(* IEC 61131-3 sources: AXOpen/src/core/ctrl/src/IxUtilities, 5 files *)

(* ---- IxCRC_16.st ---- *)
USING System.Strings;
USING System.SerDe;

NAMESPACE ix.framework.core
    FUNCTION PUBLIC IxCRC_16 : WORD
		VAR_INPUT
			In : STRING[254];
		END_VAR
		VAR
			crc : WORD := WORD#16#FFFF;
			i : UINT;
			maxIndex : UINT;
			serialized : ARRAY[0..255] OF BYTE;
		END_VAR
		VAR
			//Precalculated values for polynomial generator of value 0x1021
			CRC_TABLE : ARRAY[0..255] OF WORD := [
				WORD#16#0000, WORD#16#1021, WORD#16#2042, WORD#16#3063, WORD#16#4084, WORD#16#50A5, WORD#16#60C6, WORD#16#70E7, WORD#16#8108, WORD#16#9129, WORD#16#A14A, WORD#16#B16B, WORD#16#C18C, WORD#16#D1AD, WORD#16#E1CE, WORD#16#F1EF,
				WORD#16#1231, WORD#16#0210, WORD#16#3273, WORD#16#2252, WORD#16#52B5, WORD#16#4294, WORD#16#72F7, WORD#16#62D6, WORD#16#9339, WORD#16#8318, WORD#16#B37B, WORD#16#A35A, WORD#16#D3BD, WORD#16#C39C, WORD#16#F3FF, WORD#16#E3DE,
				WORD#16#2462, WORD#16#3443, WORD#16#0420, WORD#16#1401, WORD#16#64E6, WORD#16#74C7, WORD#16#44A4, WORD#16#5485, WORD#16#A56A, WORD#16#B54B, WORD#16#8528, WORD#16#9509, WORD#16#E5EE, WORD#16#F5CF, WORD#16#C5AC, WORD#16#D58D,
				WORD#16#3653, WORD#16#2672, WORD#16#1611, WORD#16#0630, WORD#16#76D7, WORD#16#66F6, WORD#16#5695, WORD#16#46B4, WORD#16#B75B, WORD#16#A77A, WORD#16#9719, WORD#16#8738, WORD#16#F7DF, WORD#16#E7FE, WORD#16#D79D, WORD#16#C7BC,
				WORD#16#48C4, WORD#16#58E5, WORD#16#6886, WORD#16#78A7, WORD#16#0840, WORD#16#1861, WORD#16#2802, WORD#16#3823, WORD#16#C9CC, WORD#16#D9ED, WORD#16#E98E, WORD#16#F9AF, WORD#16#8948, WORD#16#9969, WORD#16#A90A, WORD#16#B92B,
				WORD#16#5AF5, WORD#16#4AD4, WORD#16#7AB7, WORD#16#6A96, WORD#16#1A71, WORD#16#0A50, WORD#16#3A33, WORD#16#2A12, WORD#16#DBFD, WORD#16#CBDC, WORD#16#FBBF, WORD#16#EB9E, WORD#16#9B79, WORD#16#8B58, WORD#16#BB3B, WORD#16#AB1A,
				WORD#16#6CA6, WORD#16#7C87, WORD#16#4CE4, WORD#16#5CC5, WORD#16#2C22, WORD#16#3C03, WORD#16#0C60, WORD#16#1C41, WORD#16#EDAE, WORD#16#FD8F, WORD#16#CDEC, WORD#16#DDCD, WORD#16#AD2A, WORD#16#BD0B, WORD#16#8D68, WORD#16#9D49,
				WORD#16#7E97, WORD#16#6EB6, WORD#16#5ED5, WORD#16#4EF4, WORD#16#3E13, WORD#16#2E32, WORD#16#1E51, WORD#16#0E70, WORD#16#FF9F, WORD#16#EFBE, WORD#16#DFDD, WORD#16#CFFC, WORD#16#BF1B, WORD#16#AF3A, WORD#16#9F59, WORD#16#8F78,
				WORD#16#9188, WORD#16#81A9, WORD#16#B1CA, WORD#16#A1EB, WORD#16#D10C, WORD#16#C12D, WORD#16#F14E, WORD#16#E16F, WORD#16#1080, WORD#16#00A1, WORD#16#30C2, WORD#16#20E3, WORD#16#5004, WORD#16#4025, WORD#16#7046, WORD#16#6067,
				WORD#16#83B9, WORD#16#9398, WORD#16#A3FB, WORD#16#B3DA, WORD#16#C33D, WORD#16#D31C, WORD#16#E37F, WORD#16#F35E, WORD#16#02B1, WORD#16#1290, WORD#16#22F3, WORD#16#32D2, WORD#16#4235, WORD#16#5214, WORD#16#6277, WORD#16#7256,
				WORD#16#B5EA, WORD#16#A5CB, WORD#16#95A8, WORD#16#8589, WORD#16#F56E, WORD#16#E54F, WORD#16#D52C, WORD#16#C50D, WORD#16#34E2, WORD#16#24C3, WORD#16#14A0, WORD#16#0481, WORD#16#7466, WORD#16#6447, WORD#16#5424, WORD#16#4405,
				WORD#16#A7DB, WORD#16#B7FA, WORD#16#8799, WORD#16#97B8, WORD#16#E75F, WORD#16#F77E, WORD#16#C71D, WORD#16#D73C, WORD#16#26D3, WORD#16#36F2, WORD#16#0691, WORD#16#16B0, WORD#16#6657, WORD#16#7676, WORD#16#4615, WORD#16#5634,
				WORD#16#D94C, WORD#16#C96D, WORD#16#F90E, WORD#16#E92F, WORD#16#99C8, WORD#16#89E9, WORD#16#B98A, WORD#16#A9AB, WORD#16#5844, WORD#16#4865, WORD#16#7806, WORD#16#6827, WORD#16#18C0, WORD#16#08E1, WORD#16#3882, WORD#16#28A3,
				WORD#16#CB7D, WORD#16#DB5C, WORD#16#EB3F, WORD#16#FB1E, WORD#16#8BF9, WORD#16#9BD8, WORD#16#ABBB, WORD#16#BB9A, WORD#16#4A75, WORD#16#5A54, WORD#16#6A37, WORD#16#7A16, WORD#16#0AF1, WORD#16#1AD0, WORD#16#2AB3, WORD#16#3A92,
				WORD#16#FD2E, WORD#16#ED0F, WORD#16#DD6C, WORD#16#CD4D, WORD#16#BDAA, WORD#16#AD8B, WORD#16#9DE8, WORD#16#8DC9, WORD#16#7C26, WORD#16#6C07, WORD#16#5C64, WORD#16#4C45, WORD#16#3CA2, WORD#16#2C83, WORD#16#1CE0, WORD#16#0CC1,
				WORD#16#EF1F, WORD#16#FF3E, WORD#16#CF5D, WORD#16#DF7C, WORD#16#AF9B, WORD#16#BFBA, WORD#16#8FD9, WORD#16#9FF8, WORD#16#6E17, WORD#16#7E36, WORD#16#4E55, WORD#16#5E74, WORD#16#2E93, WORD#16#3EB2, WORD#16#0ED1, WORD#16#1EF0];
		END_VAR
		IxCRC_16 := crc;

		maxIndex := UINT#0;

		maxIndex := Serialize(UINT#0, In, serialized,System.SerDe.Endianness#Little) - UINT#1;

		IF maxIndex < UINT#1 THEN
			RETURN;
		END_IF;

		FOR i := UINT#1 TO maxIndex BY UINT#1 DO
			// crc := SHL(crc, 8) XOR CRC_TABLE[SHR(crc, 8) XOR bByte];
			crc := ixXor(SHL(crc, UINT#8),CRC_TABLE[TO_INT(ixXor(SHR(crc, UINT#8) , serialized[i]))]);
		END_FOR;

		IxCRC_16 := crc;
    END_FUNCTION
END_NAMESPACE

(* ---- IxCRC_32.st ---- *)
USING System.Strings;
USING System.SerDe;

NAMESPACE ix.framework.core
    FUNCTION PUBLIC IxCRC_32 : DWORD
		VAR_INPUT
			In : STRING[254];
		END_VAR
		VAR
			crc : DWORD := DWORD#16#FFFFFFFF;
			i : UINT;
			maxIndex : UINT;
			serialized : ARRAY[0..255] OF BYTE;
		END_VAR
		VAR
			//Precalculated values for polynomial generator of value 0x04C11DB7
			CRC_TABLE : ARRAY[0..255] OF DWORD := [
				DWORD#16#00000000, DWORD#16#04C11DB7, DWORD#16#09823B6E, DWORD#16#0D4326D9, DWORD#16#130476DC, DWORD#16#17C56B6B, DWORD#16#1A864DB2, DWORD#16#1E475005, DWORD#16#2608EDB8, DWORD#16#22C9F00F, DWORD#16#2F8AD6D6, DWORD#16#2B4BCB61, DWORD#16#350C9B64, DWORD#16#31CD86D3, DWORD#16#3C8EA00A, DWORD#16#384FBDBD,
				DWORD#16#4C11DB70, DWORD#16#48D0C6C7, DWORD#16#4593E01E, DWORD#16#4152FDA9, DWORD#16#5F15ADAC, DWORD#16#5BD4B01B, DWORD#16#569796C2, DWORD#16#52568B75, DWORD#16#6A1936C8, DWORD#16#6ED82B7F, DWORD#16#639B0DA6, DWORD#16#675A1011, DWORD#16#791D4014, DWORD#16#7DDC5DA3, DWORD#16#709F7B7A, DWORD#16#745E66CD,
				DWORD#16#9823B6E0, DWORD#16#9CE2AB57, DWORD#16#91A18D8E, DWORD#16#95609039, DWORD#16#8B27C03C, DWORD#16#8FE6DD8B, DWORD#16#82A5FB52, DWORD#16#8664E6E5, DWORD#16#BE2B5B58, DWORD#16#BAEA46EF, DWORD#16#B7A96036, DWORD#16#B3687D81, DWORD#16#AD2F2D84, DWORD#16#A9EE3033, DWORD#16#A4AD16EA, DWORD#16#A06C0B5D,
				DWORD#16#D4326D90, DWORD#16#D0F37027, DWORD#16#DDB056FE, DWORD#16#D9714B49, DWORD#16#C7361B4C, DWORD#16#C3F706FB, DWORD#16#CEB42022, DWORD#16#CA753D95, DWORD#16#F23A8028, DWORD#16#F6FB9D9F, DWORD#16#FBB8BB46, DWORD#16#FF79A6F1, DWORD#16#E13EF6F4, DWORD#16#E5FFEB43, DWORD#16#E8BCCD9A, DWORD#16#EC7DD02D,
				DWORD#16#34867077, DWORD#16#30476DC0, DWORD#16#3D044B19, DWORD#16#39C556AE, DWORD#16#278206AB, DWORD#16#23431B1C, DWORD#16#2E003DC5, DWORD#16#2AC12072, DWORD#16#128E9DCF, DWORD#16#164F8078, DWORD#16#1B0CA6A1, DWORD#16#1FCDBB16, DWORD#16#018AEB13, DWORD#16#054BF6A4, DWORD#16#0808D07D, DWORD#16#0CC9CDCA,
				DWORD#16#7897AB07, DWORD#16#7C56B6B0, DWORD#16#71159069, DWORD#16#75D48DDE, DWORD#16#6B93DDDB, DWORD#16#6F52C06C, DWORD#16#6211E6B5, DWORD#16#66D0FB02, DWORD#16#5E9F46BF, DWORD#16#5A5E5B08, DWORD#16#571D7DD1, DWORD#16#53DC6066, DWORD#16#4D9B3063, DWORD#16#495A2DD4, DWORD#16#44190B0D, DWORD#16#40D816BA,
				DWORD#16#ACA5C697, DWORD#16#A864DB20, DWORD#16#A527FDF9, DWORD#16#A1E6E04E, DWORD#16#BFA1B04B, DWORD#16#BB60ADFC, DWORD#16#B6238B25, DWORD#16#B2E29692, DWORD#16#8AAD2B2F, DWORD#16#8E6C3698, DWORD#16#832F1041, DWORD#16#87EE0DF6, DWORD#16#99A95DF3, DWORD#16#9D684044, DWORD#16#902B669D, DWORD#16#94EA7B2A,
				DWORD#16#E0B41DE7, DWORD#16#E4750050, DWORD#16#E9362689, DWORD#16#EDF73B3E, DWORD#16#F3B06B3B, DWORD#16#F771768C, DWORD#16#FA325055, DWORD#16#FEF34DE2, DWORD#16#C6BCF05F, DWORD#16#C27DEDE8, DWORD#16#CF3ECB31, DWORD#16#CBFFD686, DWORD#16#D5B88683, DWORD#16#D1799B34, DWORD#16#DC3ABDED, DWORD#16#D8FBA05A,
				DWORD#16#690CE0EE, DWORD#16#6DCDFD59, DWORD#16#608EDB80, DWORD#16#644FC637, DWORD#16#7A089632, DWORD#16#7EC98B85, DWORD#16#738AAD5C, DWORD#16#774BB0EB, DWORD#16#4F040D56, DWORD#16#4BC510E1, DWORD#16#46863638, DWORD#16#42472B8F, DWORD#16#5C007B8A, DWORD#16#58C1663D, DWORD#16#558240E4, DWORD#16#51435D53,
				DWORD#16#251D3B9E, DWORD#16#21DC2629, DWORD#16#2C9F00F0, DWORD#16#285E1D47, DWORD#16#36194D42, DWORD#16#32D850F5, DWORD#16#3F9B762C, DWORD#16#3B5A6B9B, DWORD#16#0315D626, DWORD#16#07D4CB91, DWORD#16#0A97ED48, DWORD#16#0E56F0FF, DWORD#16#1011A0FA, DWORD#16#14D0BD4D, DWORD#16#19939B94, DWORD#16#1D528623,
				DWORD#16#F12F560E, DWORD#16#F5EE4BB9, DWORD#16#F8AD6D60, DWORD#16#FC6C70D7, DWORD#16#E22B20D2, DWORD#16#E6EA3D65, DWORD#16#EBA91BBC, DWORD#16#EF68060B, DWORD#16#D727BBB6, DWORD#16#D3E6A601, DWORD#16#DEA580D8, DWORD#16#DA649D6F, DWORD#16#C423CD6A, DWORD#16#C0E2D0DD, DWORD#16#CDA1F604, DWORD#16#C960EBB3,
				DWORD#16#BD3E8D7E, DWORD#16#B9FF90C9, DWORD#16#B4BCB610, DWORD#16#B07DABA7, DWORD#16#AE3AFBA2, DWORD#16#AAFBE615, DWORD#16#A7B8C0CC, DWORD#16#A379DD7B, DWORD#16#9B3660C6, DWORD#16#9FF77D71, DWORD#16#92B45BA8, DWORD#16#9675461F, DWORD#16#8832161A, DWORD#16#8CF30BAD, DWORD#16#81B02D74, DWORD#16#857130C3,
				DWORD#16#5D8A9099, DWORD#16#594B8D2E, DWORD#16#5408ABF7, DWORD#16#50C9B640, DWORD#16#4E8EE645, DWORD#16#4A4FFBF2, DWORD#16#470CDD2B, DWORD#16#43CDC09C, DWORD#16#7B827D21, DWORD#16#7F436096, DWORD#16#7200464F, DWORD#16#76C15BF8, DWORD#16#68860BFD, DWORD#16#6C47164A, DWORD#16#61043093, DWORD#16#65C52D24,
				DWORD#16#119B4BE9, DWORD#16#155A565E, DWORD#16#18197087, DWORD#16#1CD86D30, DWORD#16#029F3D35, DWORD#16#065E2082, DWORD#16#0B1D065B, DWORD#16#0FDC1BEC, DWORD#16#3793A651, DWORD#16#3352BBE6, DWORD#16#3E119D3F, DWORD#16#3AD08088, DWORD#16#2497D08D, DWORD#16#2056CD3A, DWORD#16#2D15EBE3, DWORD#16#29D4F654,
				DWORD#16#C5A92679, DWORD#16#C1683BCE, DWORD#16#CC2B1D17, DWORD#16#C8EA00A0, DWORD#16#D6AD50A5, DWORD#16#D26C4D12, DWORD#16#DF2F6BCB, DWORD#16#DBEE767C, DWORD#16#E3A1CBC1, DWORD#16#E760D676, DWORD#16#EA23F0AF, DWORD#16#EEE2ED18, DWORD#16#F0A5BD1D, DWORD#16#F464A0AA, DWORD#16#F9278673, DWORD#16#FDE69BC4,
				DWORD#16#89B8FD09, DWORD#16#8D79E0BE, DWORD#16#803AC667, DWORD#16#84FBDBD0, DWORD#16#9ABC8BD5, DWORD#16#9E7D9662, DWORD#16#933EB0BB, DWORD#16#97FFAD0C, DWORD#16#AFB010B1, DWORD#16#AB710D06, DWORD#16#A6322BDF, DWORD#16#A2F33668, DWORD#16#BCB4666D, DWORD#16#B8757BDA, DWORD#16#B5365D03, DWORD#16#B1F740B4];
		END_VAR
		IxCRC_32 := crc;

		maxIndex := UINT#0;

		maxIndex := Serialize(UINT#0, In, serialized,System.SerDe.Endianness#Little) - UINT#1;

		IF maxIndex < UINT#1 THEN
			RETURN;
		END_IF;

		FOR i := UINT#1 TO maxIndex BY UINT#1 DO
			// posD := SHR(crc, 24) XOR bByte;
			// pos := UDINT_TO_BYTE(posD);

			// crc := SHL(crc, 8) XOR CRC_TABLE[pos];

			crc := ixXor(SHL(crc, UINT#8),CRC_TABLE[TO_INT(ixXor(SHR(crc, UINT#24) , serialized[i]))]);
		END_FOR;

		IxCRC_32 := crc;
    END_FUNCTION
END_NAMESPACE

(* ---- IxCRC_8.st ---- *)
USING System.Strings;
USING System.SerDe;

NAMESPACE ix.framework.core
    FUNCTION PUBLIC IxCRC_8 : BYTE
		VAR_INPUT
			In : STRING[254];
		END_VAR
		VAR
			crc : BYTE := BYTE#16#FF;
			i : UINT;
			maxIndex : UINT;
			serialized : ARRAY[0..255] OF BYTE;
		END_VAR
		VAR
			//Precalculated values for polynomial generator of value 0x1D
			CRC_TABLE : ARRAY[0..255] OF BYTE := [
				BYTE#16#00,	BYTE#16#1D,	BYTE#16#3A,	BYTE#16#27,	BYTE#16#74,	BYTE#16#69,	BYTE#16#4E,	BYTE#16#53,	BYTE#16#E8,	BYTE#16#F5,	BYTE#16#D2,	BYTE#16#CF,	BYTE#16#9C,	BYTE#16#81,	BYTE#16#A6,	BYTE#16#BB,
				BYTE#16#CD,	BYTE#16#D0,	BYTE#16#F7,	BYTE#16#EA,	BYTE#16#B9,	BYTE#16#A4,	BYTE#16#83,	BYTE#16#9E,	BYTE#16#25,	BYTE#16#38,	BYTE#16#1F,	BYTE#16#02,	BYTE#16#51,	BYTE#16#4C,	BYTE#16#6B,	BYTE#16#76,
				BYTE#16#87,	BYTE#16#9A,	BYTE#16#BD,	BYTE#16#A0,	BYTE#16#F3,	BYTE#16#EE,	BYTE#16#C9,	BYTE#16#D4,	BYTE#16#6F,	BYTE#16#72,	BYTE#16#55,	BYTE#16#48,	BYTE#16#1B,	BYTE#16#06,	BYTE#16#21,	BYTE#16#3C,
				BYTE#16#4A,	BYTE#16#57,	BYTE#16#70,	BYTE#16#6D,	BYTE#16#3E,	BYTE#16#23,	BYTE#16#04,	BYTE#16#19,	BYTE#16#A2,	BYTE#16#BF,	BYTE#16#98,	BYTE#16#85,	BYTE#16#D6,	BYTE#16#CB,	BYTE#16#EC,	BYTE#16#F1,
				BYTE#16#13,	BYTE#16#0E,	BYTE#16#29,	BYTE#16#34,	BYTE#16#67,	BYTE#16#7A,	BYTE#16#5D,	BYTE#16#40,	BYTE#16#FB,	BYTE#16#E6,	BYTE#16#C1,	BYTE#16#DC,	BYTE#16#8F,	BYTE#16#92,	BYTE#16#B5,	BYTE#16#A8,
				BYTE#16#DE,	BYTE#16#C3,	BYTE#16#E4,	BYTE#16#F9,	BYTE#16#AA,	BYTE#16#B7,	BYTE#16#90,	BYTE#16#8D,	BYTE#16#36,	BYTE#16#2B,	BYTE#16#0C,	BYTE#16#11,	BYTE#16#42,	BYTE#16#5F,	BYTE#16#78,	BYTE#16#65,
				BYTE#16#94,	BYTE#16#89,	BYTE#16#AE,	BYTE#16#B3,	BYTE#16#E0,	BYTE#16#FD,	BYTE#16#DA,	BYTE#16#C7,	BYTE#16#7C,	BYTE#16#61,	BYTE#16#46,	BYTE#16#5B,	BYTE#16#08,	BYTE#16#15,	BYTE#16#32,	BYTE#16#2F,
				BYTE#16#59,	BYTE#16#44,	BYTE#16#63,	BYTE#16#7E,	BYTE#16#2D,	BYTE#16#30,	BYTE#16#17,	BYTE#16#0A,	BYTE#16#B1,	BYTE#16#AC,	BYTE#16#8B,	BYTE#16#96,	BYTE#16#C5,	BYTE#16#D8,	BYTE#16#FF,	BYTE#16#E2,
				BYTE#16#26,	BYTE#16#3B,	BYTE#16#1C,	BYTE#16#01,	BYTE#16#52,	BYTE#16#4F,	BYTE#16#68,	BYTE#16#75,	BYTE#16#CE,	BYTE#16#D3,	BYTE#16#F4,	BYTE#16#E9,	BYTE#16#BA,	BYTE#16#A7,	BYTE#16#80,	BYTE#16#9D,
				BYTE#16#EB,	BYTE#16#F6,	BYTE#16#D1,	BYTE#16#CC,	BYTE#16#9F,	BYTE#16#82,	BYTE#16#A5,	BYTE#16#B8,	BYTE#16#03,	BYTE#16#1E,	BYTE#16#39,	BYTE#16#24,	BYTE#16#77,	BYTE#16#6A,	BYTE#16#4D,	BYTE#16#50,
				BYTE#16#A1,	BYTE#16#BC,	BYTE#16#9B,	BYTE#16#86,	BYTE#16#D5,	BYTE#16#C8,	BYTE#16#EF,	BYTE#16#F2,	BYTE#16#49,	BYTE#16#54,	BYTE#16#73,	BYTE#16#6E,	BYTE#16#3D,	BYTE#16#20,	BYTE#16#07,	BYTE#16#1A,
				BYTE#16#6C,	BYTE#16#71,	BYTE#16#56,	BYTE#16#4B,	BYTE#16#18,	BYTE#16#05,	BYTE#16#22,	BYTE#16#3F,	BYTE#16#84,	BYTE#16#99,	BYTE#16#BE,	BYTE#16#A3,	BYTE#16#F0,	BYTE#16#ED,	BYTE#16#CA,	BYTE#16#D7,
				BYTE#16#35,	BYTE#16#28,	BYTE#16#0F,	BYTE#16#12,	BYTE#16#41,	BYTE#16#5C,	BYTE#16#7B,	BYTE#16#66,	BYTE#16#DD,	BYTE#16#C0,	BYTE#16#E7,	BYTE#16#FA,	BYTE#16#A9,	BYTE#16#B4,	BYTE#16#93,	BYTE#16#8E,
				BYTE#16#F8,	BYTE#16#E5,	BYTE#16#C2,	BYTE#16#DF,	BYTE#16#8C,	BYTE#16#91,	BYTE#16#B6,	BYTE#16#AB,	BYTE#16#10,	BYTE#16#0D,	BYTE#16#2A,	BYTE#16#37,	BYTE#16#64,	BYTE#16#79,	BYTE#16#5E,	BYTE#16#43,
				BYTE#16#B2,	BYTE#16#AF,	BYTE#16#88,	BYTE#16#95,	BYTE#16#C6,	BYTE#16#DB,	BYTE#16#FC,	BYTE#16#E1,	BYTE#16#5A,	BYTE#16#47,	BYTE#16#60,	BYTE#16#7D,	BYTE#16#2E,	BYTE#16#33,	BYTE#16#14,	BYTE#16#09,
				BYTE#16#7F,	BYTE#16#62,	BYTE#16#45,	BYTE#16#58,	BYTE#16#0B,	BYTE#16#16,	BYTE#16#31,	BYTE#16#2C,	BYTE#16#97,	BYTE#16#8A,	BYTE#16#AD,	BYTE#16#B0,	BYTE#16#E3,	BYTE#16#FE,	BYTE#16#D9,	BYTE#16#C4];
		END_VAR
		IxCRC_8 := crc;

		maxIndex := UINT#0;

		maxIndex := Serialize(UINT#0, In, serialized, System.SerDe.Endianness#Little) - UINT#1;

		IF maxIndex < UINT#1 THEN
			RETURN;
		END_IF;

		FOR i := UINT#1 TO maxIndex BY UINT#1 DO
			//crc := CRC_TABLE[bByte XOR crc];
			crc := CRC_TABLE[TO_INT(ixXor(crc , TO_BYTE(TO_CHAR(serialized[i]))))];
		END_FOR;
		IxCRC_8 := crc;
    END_FUNCTION
END_NAMESPACE

(* ---- XORs.st ---- *)
// USING System.BitAccess;

NAMESPACE ix.framework.core
    FUNCTION ixXor : BYTE
        VAR_INPUT
            In1 : BYTE;
            In2 : BYTE;
        END_VAR
        VAR_TEMP
            retval : BYTE;
            i : USINT;
        END_VAR
        retval := BYTE#0;

        // TODO check the performance of both principles
        // FOR i := USINT#0 TO USINT#7 DO
        //     SetBit(retval,i,GetBit(In1,i) XOR GetBit(In2,i));
        // END_FOR;

        retval.%X0 := In1.%X0  XOR In2.%X0 ;
        retval.%X1 := In1.%X1  XOR In2.%X1 ;
        retval.%X2 := In1.%X2  XOR In2.%X2 ;
        retval.%X3 := In1.%X3  XOR In2.%X3 ;
        retval.%X4 := In1.%X4  XOR In2.%X4 ;
        retval.%X5 := In1.%X5  XOR In2.%X5 ;
        retval.%X6 := In1.%X6  XOR In2.%X6 ;
        retval.%X7 := In1.%X7  XOR In2.%X7 ;

        ixXor := retval;
    END_FUNCTION

    FUNCTION ixXor : WORD
        VAR_INPUT
            In1 : WORD;
            In2 : WORD;
        END_VAR
        VAR_TEMP
            retval : WORD;
            i : USINT;
        END_VAR
        retval := WORD#0;

        // TODO check the performance of both principles
        // FOR i := USINT#0 TO USINT#15 DO
        //     SetBit(retval,i,GetBit(In1,i) XOR GetBit(In2,i));
        // END_FOR;

        retval.%X0  := In1.%X0   XOR In2.%X0  ;
        retval.%X1  := In1.%X1   XOR In2.%X1  ;
        retval.%X2  := In1.%X2   XOR In2.%X2  ;
        retval.%X3  := In1.%X3   XOR In2.%X3  ;
        retval.%X4  := In1.%X4   XOR In2.%X4  ;
        retval.%X5  := In1.%X5   XOR In2.%X5  ;
        retval.%X6  := In1.%X6   XOR In2.%X6  ;
        retval.%X7  := In1.%X7   XOR In2.%X7  ;
        retval.%X8  := In1.%X8   XOR In2.%X8  ;
        retval.%X9  := In1.%X9   XOR In2.%X9  ;
        retval.%X10 := In1.%X10  XOR In2.%X10 ;
        retval.%X11 := In1.%X11  XOR In2.%X11 ;
        retval.%X12 := In1.%X12  XOR In2.%X12 ;
        retval.%X13 := In1.%X13  XOR In2.%X13 ;
        retval.%X14 := In1.%X14  XOR In2.%X14 ;
        retval.%X15 := In1.%X15  XOR In2.%X15 ;

        ixXor := retval;
    END_FUNCTION

    FUNCTION ixXor : DWORD
        VAR_INPUT
            In1 : DWORD;
            In2 : DWORD;
        END_VAR
        VAR_TEMP
            retval : DWORD;
            i : USINT;
        END_VAR
        retval := DWORD#0;

        // TODO check the performance of both principles
        // FOR i := USINT#0 TO USINT#31 DO
        //     SetBit(retval,i,GetBit(In1,i) XOR GetBit(In2,i));
        // END_FOR;

        retval.%X0  := In1.%X0   XOR In2.%X0  ;
        retval.%X1  := In1.%X1   XOR In2.%X1  ;
        retval.%X2  := In1.%X2   XOR In2.%X2  ;
        retval.%X3  := In1.%X3   XOR In2.%X3  ;
        retval.%X4  := In1.%X4   XOR In2.%X4  ;
        retval.%X5  := In1.%X5   XOR In2.%X5  ;
        retval.%X6  := In1.%X6   XOR In2.%X6  ;
        retval.%X7  := In1.%X7   XOR In2.%X7  ;
        retval.%X8  := In1.%X8   XOR In2.%X8  ;
        retval.%X9  := In1.%X9   XOR In2.%X9  ;
        retval.%X10 := In1.%X10  XOR In2.%X10 ;
        retval.%X11 := In1.%X11  XOR In2.%X11 ;
        retval.%X12 := In1.%X12  XOR In2.%X12 ;
        retval.%X13 := In1.%X13  XOR In2.%X13 ;
        retval.%X14 := In1.%X14  XOR In2.%X14 ;
        retval.%X15 := In1.%X15  XOR In2.%X15 ;
        retval.%X16 := In1.%X16  XOR In2.%X16 ;
        retval.%X17 := In1.%X17  XOR In2.%X17 ;
        retval.%X18 := In1.%X18  XOR In2.%X18 ;
        retval.%X19 := In1.%X19  XOR In2.%X19 ;
        retval.%X20 := In1.%X20  XOR In2.%X20 ;
        retval.%X21 := In1.%X21  XOR In2.%X21 ;
        retval.%X22 := In1.%X22  XOR In2.%X22 ;
        retval.%X23 := In1.%X23  XOR In2.%X23 ;
        retval.%X24 := In1.%X24  XOR In2.%X24 ;
        retval.%X25 := In1.%X25  XOR In2.%X25 ;
        retval.%X26 := In1.%X26  XOR In2.%X26 ;
        retval.%X27 := In1.%X27  XOR In2.%X27 ;
        retval.%X28 := In1.%X28  XOR In2.%X28 ;
        retval.%X29 := In1.%X29  XOR In2.%X29 ;
        retval.%X30 := In1.%X30  XOR In2.%X30 ;
        retval.%X31 := In1.%X31  XOR In2.%X31 ;
        ixXor := retval;
    END_FUNCTION

    FUNCTION ixXor : LWORD
        VAR_INPUT
            In1 : LWORD;
            In2 : LWORD;
        END_VAR
        VAR_TEMP
            retval : LWORD;
            i : USINT;
        END_VAR
        retval := LWORD#0;

        // TODO check the performance of both principles
        // FOR i := USINT#0 TO USINT#63 DO
        //     SetBit(retval,i,GetBit(In1,i) XOR GetBit(In2,i));
        // END_FOR;

        retval.%X0  := In1.%X0   XOR In2.%X0  ;
        retval.%X1  := In1.%X1   XOR In2.%X1  ;
        retval.%X2  := In1.%X2   XOR In2.%X2  ;
        retval.%X3  := In1.%X3   XOR In2.%X3  ;
        retval.%X4  := In1.%X4   XOR In2.%X4  ;
        retval.%X5  := In1.%X5   XOR In2.%X5  ;
        retval.%X6  := In1.%X6   XOR In2.%X6  ;
        retval.%X7  := In1.%X7   XOR In2.%X7  ;
        retval.%X8  := In1.%X8   XOR In2.%X8  ;
        retval.%X9  := In1.%X9   XOR In2.%X9  ;
        retval.%X10 := In1.%X10  XOR In2.%X10 ;
        retval.%X11 := In1.%X11  XOR In2.%X11 ;
        retval.%X12 := In1.%X12  XOR In2.%X12 ;
        retval.%X13 := In1.%X13  XOR In2.%X13 ;
        retval.%X14 := In1.%X14  XOR In2.%X14 ;
        retval.%X15 := In1.%X15  XOR In2.%X15 ;
        retval.%X16 := In1.%X16  XOR In2.%X16 ;
        retval.%X17 := In1.%X17  XOR In2.%X17 ;
        retval.%X18 := In1.%X18  XOR In2.%X18 ;
        retval.%X19 := In1.%X19  XOR In2.%X19 ;
        retval.%X20 := In1.%X20  XOR In2.%X20 ;
        retval.%X21 := In1.%X21  XOR In2.%X21 ;
        retval.%X22 := In1.%X22  XOR In2.%X22 ;
        retval.%X23 := In1.%X23  XOR In2.%X23 ;
        retval.%X24 := In1.%X24  XOR In2.%X24 ;
        retval.%X25 := In1.%X25  XOR In2.%X25 ;
        retval.%X26 := In1.%X26  XOR In2.%X26 ;
        retval.%X27 := In1.%X27  XOR In2.%X27 ;
        retval.%X28 := In1.%X28  XOR In2.%X28 ;
        retval.%X29 := In1.%X29  XOR In2.%X29 ;
        retval.%X30 := In1.%X30  XOR In2.%X30 ;
        retval.%X31 := In1.%X31  XOR In2.%X31 ;
        retval.%X32 := In1.%X32  XOR In2.%X32 ;
        retval.%X33 := In1.%X33  XOR In2.%X33 ;
        retval.%X34 := In1.%X34  XOR In2.%X34 ;
        retval.%X35 := In1.%X35  XOR In2.%X35 ;
        retval.%X36 := In1.%X36  XOR In2.%X36 ;
        retval.%X37 := In1.%X37  XOR In2.%X37 ;
        retval.%X38 := In1.%X38  XOR In2.%X38 ;
        retval.%X39 := In1.%X39  XOR In2.%X39 ;
        retval.%X40 := In1.%X40  XOR In2.%X40 ;
        retval.%X41 := In1.%X41  XOR In2.%X41 ;
        retval.%X42 := In1.%X42  XOR In2.%X42 ;
        retval.%X43 := In1.%X43  XOR In2.%X43 ;
        retval.%X44 := In1.%X44  XOR In2.%X44 ;
        retval.%X45 := In1.%X45  XOR In2.%X45 ;
        retval.%X46 := In1.%X46  XOR In2.%X46 ;
        retval.%X47 := In1.%X47  XOR In2.%X47 ;
        retval.%X48 := In1.%X48  XOR In2.%X48 ;
        retval.%X49 := In1.%X49  XOR In2.%X49 ;
        retval.%X50 := In1.%X50  XOR In2.%X50 ;
        retval.%X51 := In1.%X51  XOR In2.%X51 ;
        retval.%X52 := In1.%X52  XOR In2.%X52 ;
        retval.%X53 := In1.%X53  XOR In2.%X53 ;
        retval.%X54 := In1.%X54  XOR In2.%X54 ;
        retval.%X55 := In1.%X55  XOR In2.%X55 ;
        retval.%X56 := In1.%X56  XOR In2.%X56 ;
        retval.%X57 := In1.%X57  XOR In2.%X57 ;
        retval.%X58 := In1.%X58  XOR In2.%X58 ;
        retval.%X59 := In1.%X59  XOR In2.%X59 ;
        retval.%X60 := In1.%X60  XOR In2.%X60 ;
        retval.%X61 := In1.%X61  XOR In2.%X61 ;
        retval.%X62 := In1.%X62  XOR In2.%X62 ;
        retval.%X63 := In1.%X63  XOR In2.%X63 ;
        ixXor := retval;
    END_FUNCTION
END_NAMESPACE

(* ---- StringBuilder.st ---- *)
USING System.Strings;

NAMESPACE ix.framework.core
	/// <summary>
	/// Allows to concat strings using fluent interface. It's similar to C# StringBuilder class
	/// Usage as follows :
	/// <code>
	/// 	ErrorString := _stringBuilder
	/// 		.Clear()
	/// 		.Append('Error number: ')
	/// 		.Append(ErrorNumber)
	/// 		.Append('. Message: ')
	/// 		.Append(ErrorMessage)
	/// 		.Append('.')
	/// 		.AsString();
	/// </code>
	/// Inspired by Gerhard Barteling blogpost at https://www.plccoder.com/fluent-code/
	/// </summary>
    CLASS PUBLIC StringBuilder
		VAR
            _workString: STRING[254];
        END_VAR

		METHOD PUBLIC Clear : REF_TO StringBuilder
			_workString := '';
			Clear ?= REF(THIS);
		END_METHOD

		METHOD PUBLIC Append : REF_TO StringBuilder
			VAR_INPUT
				Data : BOOL;
			END_VAR
			_workString := Concat(_workString,ToString(Data));
			Append ?= REF(THIS);
		END_METHOD

		METHOD PUBLIC Append : REF_TO StringBuilder
			VAR_INPUT
				Data : BYTE;
			END_VAR
			_workString := Concat(_workString,ToString(Data));
			Append ?= REF(THIS);
		END_METHOD

		METHOD PUBLIC Append : REF_TO StringBuilder
			VAR_INPUT
				Data : WORD;
			END_VAR
			_workString := Concat(_workString,ToString(Data));
			Append ?= REF(THIS);
		END_METHOD

		METHOD PUBLIC Append : REF_TO StringBuilder
			VAR_INPUT
				Data : DWORD;
			END_VAR
			_workString := Concat(_workString,ToString(Data));
			Append ?= REF(THIS);
		END_METHOD

		METHOD PUBLIC Append : REF_TO StringBuilder
			VAR_INPUT
				Data : LWORD;
			END_VAR
			_workString := Concat(_workString,ToString(Data));
			Append ?= REF(THIS);
		END_METHOD

		METHOD PUBLIC Append : REF_TO StringBuilder
			VAR_INPUT
				Data : SINT;
			END_VAR
			_workString := Concat(_workString,ToString(Data));
			Append ?= REF(THIS);
		END_METHOD

		METHOD PUBLIC Append : REF_TO StringBuilder
			VAR_INPUT
				Data : INT;
			END_VAR
			_workString := Concat(_workString,ToString(Data));
			Append ?= REF(THIS);
		END_METHOD

		METHOD PUBLIC Append : REF_TO StringBuilder
			VAR_INPUT
				Data : DINT;
			END_VAR
			_workString := Concat(_workString,ToString(Data));
			Append ?= REF(THIS);
		END_METHOD

		METHOD PUBLIC Append : REF_TO StringBuilder
			VAR_INPUT
				Data : LINT;
			END_VAR
			_workString := Concat(_workString,ToString(Data));
			Append ?= REF(THIS);
		END_METHOD

		METHOD PUBLIC Append : REF_TO StringBuilder
			VAR_INPUT
				Data : USINT;
			END_VAR
			_workString := Concat(_workString,ToString(Data));
			Append ?= REF(THIS);
		END_METHOD

		METHOD PUBLIC Append : REF_TO StringBuilder
			VAR_INPUT
				Data : UINT;
			END_VAR
			_workString := Concat(_workString,ToString(Data));
			Append ?= REF(THIS);
		END_METHOD

		METHOD PUBLIC Append : REF_TO StringBuilder
			VAR_INPUT
				Data : UDINT;
			END_VAR
			_workString := Concat(_workString,ToString(Data));
			Append ?= REF(THIS);
		END_METHOD

		METHOD PUBLIC Append : REF_TO StringBuilder
			VAR_INPUT
				Data : ULINT;
			END_VAR
			_workString := Concat(_workString,ToString(Data));
			Append ?= REF(THIS);
		END_METHOD

		METHOD PUBLIC Append : REF_TO StringBuilder
			VAR_INPUT
				Data : REAL;
			END_VAR
			_workString := Concat(_workString,ToString(Data));
			Append ?= REF(THIS);
		END_METHOD

		METHOD PUBLIC Append : REF_TO StringBuilder
			VAR_INPUT
				Data : LREAL;
			END_VAR
			_workString := Concat(_workString,ToString(Data));
			Append ?= REF(THIS);
		END_METHOD

		METHOD PUBLIC Append : REF_TO StringBuilder
			VAR_INPUT
				Data : TIME;
			END_VAR
			_workString := Concat(_workString,ToString(Data));
			Append ?= REF(THIS);
		END_METHOD

		METHOD PUBLIC Append : REF_TO StringBuilder
			VAR_INPUT
				Data : LTIME;
			END_VAR
			_workString := Concat(_workString,ToString(Data));
			Append ?= REF(THIS);
		END_METHOD

		METHOD PUBLIC Append : REF_TO StringBuilder
			VAR_INPUT
				Data : DATE;
			END_VAR
			_workString := Concat(_workString,ToString(Data));
			Append ?= REF(THIS);
		END_METHOD

		METHOD PUBLIC Append : REF_TO StringBuilder
			VAR_INPUT
				Data : LDATE;
			END_VAR
			_workString := Concat(_workString,ToString(Data));
			Append ?= REF(THIS);
		END_METHOD

		METHOD PUBLIC Append : REF_TO StringBuilder
			VAR_INPUT
				Data : TIME_OF_DAY;
			END_VAR
			_workString := Concat(_workString,ToString(Data));
			Append ?= REF(THIS);
		END_METHOD

		METHOD PUBLIC Append : REF_TO StringBuilder
			VAR_INPUT
				Data : LTIME_OF_DAY;
			END_VAR
			_workString := Concat(_workString,ToString(Data));
			Append ?= REF(THIS);
		END_METHOD

		METHOD PUBLIC Append : REF_TO StringBuilder
			VAR_INPUT
				Data : DATE_AND_TIME;
			END_VAR
			_workString := Concat(_workString,ToString(Data));
			Append ?= REF(THIS);
		END_METHOD

		METHOD PUBLIC Append : REF_TO StringBuilder
			VAR_INPUT
				Data : LDATE_AND_TIME;
			END_VAR
			_workString := Concat(_workString,ToString(Data));
			Append ?= REF(THIS);
		END_METHOD

		METHOD PUBLIC Append : REF_TO StringBuilder
			VAR_INPUT
				Data : CHAR;
			END_VAR
			_workString := Concat(_workString,Data);
			Append ?= REF(THIS);
		END_METHOD

		// METHOD PUBLIC Append : REF_TO StringBuilder
		// 	VAR_INPUT
		// 		Data : WCHAR;
		// 	END_VAR
		// 	_workString := Concat(_workString,ToString(Data));
		// 	Append ?= REF(THIS);
		// END_METHOD

		METHOD PUBLIC Append : REF_TO StringBuilder
			VAR_INPUT
				Data :STRING[254];
			END_VAR
			_workString := Concat(_workString,Data);
			Append ?= REF(THIS);
		END_METHOD

		// METHOD PUBLIC  Append : REF_TO StringBuilder
		// 	VAR_INPUT
		// 		Data :WSTRING[254];
		// 	END_VAR
		// 	_workString := Concat(_workString,ToString(Data));
		// 	Append ?= REF(THIS);
		// END_METHOD

		METHOD PUBLIC AsString : STRING[IxIntConstants#MAX_MESSAGE_TEXT_LENGHT]
			AsString := _workString;
		END_METHOD
    END_CLASS
END_NAMESPACE
